(* PLC project prj, KAIST_DSLAB noNameNow 1, author bwkim *)
(* stored: creationDateTime 2015-7-21T04:57:15, modificationDateTime 2015-7-21T04:57:15 *)

PROGRAM program6____sub1
  VAR
    VR_PTON : null;
  END_VAR
  VAR
    VR_TON : null;
  END_VAR
  VAR_INPUT
    K_DELAY : null;
  END_VAR
  VAR_OUTPUT
    PTON_et : null;
  END_VAR
  VAR_OUTPUT
    TON_et : null;
  END_VAR
  VAR_IN_OUT
    TRIP_LOGIC : BOOL := FALSE;
  END_VAR
  VAR_IN_OUT
    PTRIP_LOGIC : BOOL := FALSE;
  END_VAR
  VAR  (* added by the conversion: wires and edge detectors of the diagram *)
    _ADD2_REAL34_OUT : ANY;
    _DIV_REAL56_OUT : INT;
    _SEL_REAL72_OUT : INT;
    _SEL_REAL73_OUT : INT;
    _SEL_REAL74_OUT : INT;
    _SEL_DINT75_OUT : BOOL;
    _SEL_REAL39_OUT : INT;
    _SEL_DINT82_OUT : BOOL;
    _SEL_DINT83_OUT : INT;
    _AND2_BOOL63_OUT : BOOL;
    _SEL_DINT86_OUT : INT;
    _SEL_DINT87_OUT : INT;
    _AND2_BOOL41_OUT : ANY;
  END_VAR

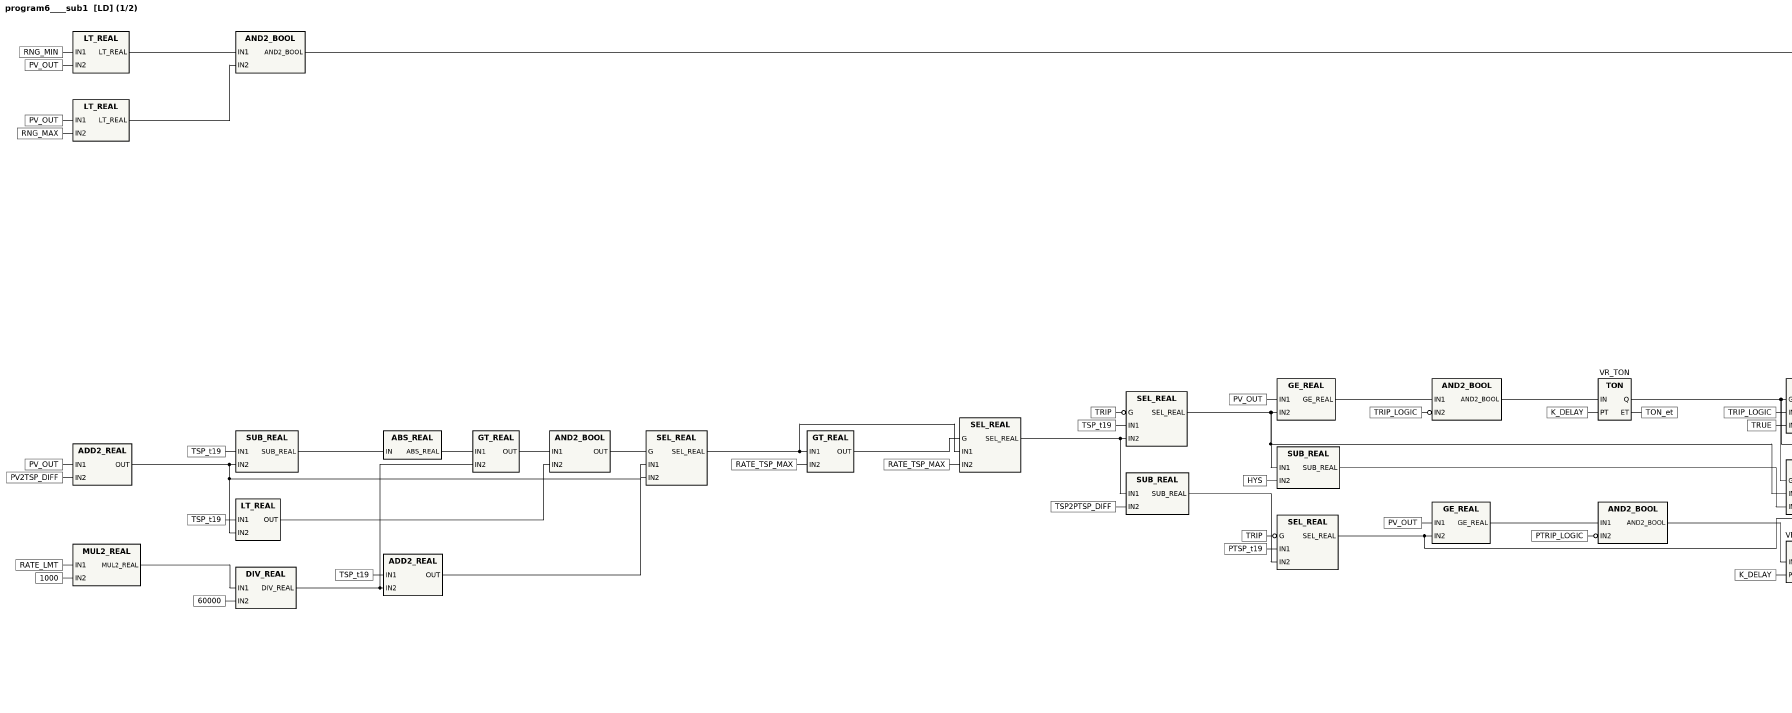
(* LD diagram, written out as Structured Text *)
_ADD2_REAL34_OUT := ADD2_REAL(PV_OUT, PV2TSP_DIFF);
_DIV_REAL56_OUT := DIV_REAL(MUL2_REAL(RATE_LMT, 1000), 60000);
_SEL_REAL72_OUT := SEL_REAL(AND2_BOOL(GT_REAL(ABS_REAL(SUB_REAL(TSP_t19, _ADD2_REAL34_OUT)), _DIV_REAL56_OUT), LT_REAL(TSP_t19, _ADD2_REAL34_OUT)), _ADD2_REAL34_OUT, ADD2_REAL(TSP_t19, _DIV_REAL56_OUT));
_SEL_REAL73_OUT := SEL_REAL(GT_REAL(_SEL_REAL72_OUT, RATE_TSP_MAX), _SEL_REAL72_OUT, RATE_TSP_MAX);
_SEL_REAL74_OUT := SEL_REAL(NOT TRIP, PTSP_t19, SUB_REAL(_SEL_REAL73_OUT, TSP2PTSP_DIFF));
VR_PTON(IN := AND2_BOOL(GE_REAL(PV_OUT, _SEL_REAL74_OUT), NOT PTRIP_LOGIC), PT := K_DELAY);
_SEL_DINT75_OUT := SEL_DINT(VR_PTON.Q, PTRIP_LOGIC, TRUE);
PTRIP_LOGIC := _SEL_DINT75_OUT;
PTON_et := VR_PTON.ET;
_SEL_REAL39_OUT := SEL_REAL(NOT TRIP, TSP_t19, _SEL_REAL73_OUT);
VR_TON(IN := AND2_BOOL(GE_REAL(PV_OUT, _SEL_REAL39_OUT), NOT TRIP_LOGIC), PT := K_DELAY);
_SEL_DINT82_OUT := SEL_DINT(VR_TON.Q, TRIP_LOGIC, TRUE);
TRIP_LOGIC := _SEL_DINT82_OUT;
TON_et := VR_TON.ET;
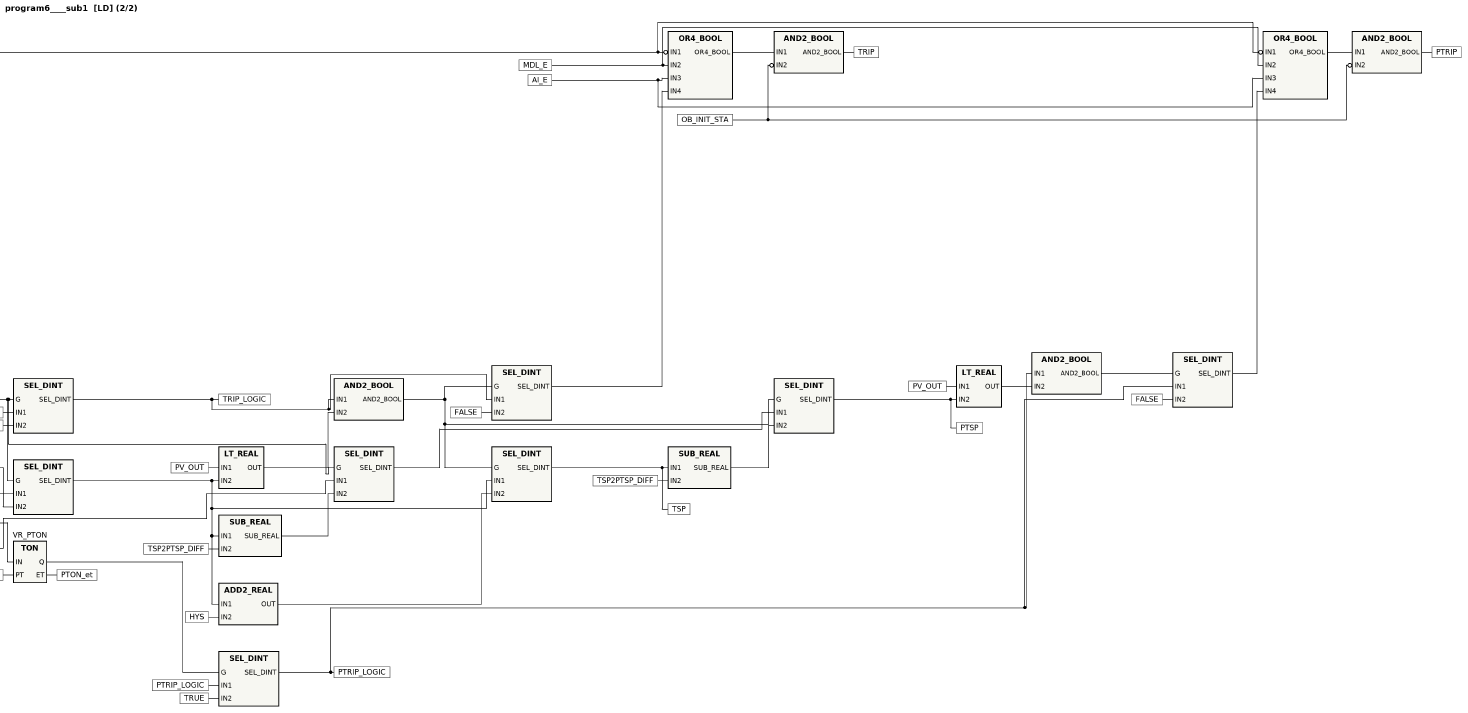
_SEL_DINT83_OUT := SEL_DINT(VR_TON.Q, _SEL_REAL39_OUT, SUB_REAL(_SEL_REAL39_OUT, HYS));
_AND2_BOOL63_OUT := AND2_BOOL(_SEL_DINT82_OUT, LT_REAL(PV_OUT, _SEL_DINT83_OUT));
_SEL_DINT86_OUT := SEL_DINT(_AND2_BOOL63_OUT, _SEL_DINT83_OUT, ADD2_REAL(_SEL_DINT83_OUT, HYS));
TSP := _SEL_DINT86_OUT;
_SEL_DINT87_OUT := SEL_DINT(_AND2_BOOL63_OUT, SEL_DINT(VR_TON.Q, _SEL_REAL74_OUT, SUB_REAL(_SEL_DINT83_OUT, TSP2PTSP_DIFF)), SUB_REAL(_SEL_DINT86_OUT, TSP2PTSP_DIFF));
PTSP := _SEL_DINT87_OUT;
_AND2_BOOL41_OUT := AND2_BOOL(LT_REAL(RNG_MIN, PV_OUT), LT_REAL(PV_OUT, RNG_MAX));
PTRIP := AND2_BOOL(OR4_BOOL(NOT _AND2_BOOL41_OUT, MDL_E, AI_E, SEL_DINT(AND2_BOOL(_SEL_DINT75_OUT, LT_REAL(PV_OUT, _SEL_DINT87_OUT)), _SEL_DINT75_OUT, FALSE)), NOT OB_INIT_STA);
TRIP := AND2_BOOL(OR4_BOOL(NOT _AND2_BOOL41_OUT, MDL_E, AI_E, SEL_DINT(_AND2_BOOL63_OUT, _SEL_DINT82_OUT, FALSE)), NOT OB_INIT_STA);
END_PROGRAM
